(* Logix 5000 project; controller WWTP_SOLIDS_CLX vendor 1 type 14 code 54 rev 17.2; software revision 17.00; part 15 of 16 *)
(* tags used below, declared in another part *)
   Equip_Torque : ALIAS FOR I_SolidsTkDrive_Torque;
   Equip_Torque_IOFault : ALIAS FOR I_SolidsTkDrive_Torque_IOFault;
   I_P600_Fault : ALIAS FOR Local:3:I.DATA.1;
   I_P600_Fault_IOFault : ALIAS FOR Local:3:I.Fault.1;
   I_P600_InAuto : ALIAS FOR Local:3:I.Data.4;
   I_P600_InAuto_IOFault : ALIAS FOR Local:3:I.Fault.4;
   I_P600_RunFdbk : ALIAS FOR Local:3:I.Data.2;
   I_P600_RunFdbk_IOFault : ALIAS FOR Local:3:I.Fault.2;
   I_P602_Fault : ALIAS FOR Local:3:I.Data.9;
   I_P602_Fault_IOFault : ALIAS FOR Local:3:I.Fault.9;
   I_P602_InAuto : ALIAS FOR Local:3:I.Data.7;
   I_P602_InAuto_IOFault : ALIAS FOR Local:3:I.Fault.7;
   I_P602_RunFdbk : ALIAS FOR Local:3:I.Data.8;
   I_P602_RunFdbk_IOFault : ALIAS FOR Local:3:I.Fault.8;
   I_PV600_CloseLS : ALIAS FOR Local:3:I.Data.14;
   I_PV600_CloseLS_IOFault : ALIAS FOR Local:3:I.Fault.14;
   I_PV600_InAuto : ALIAS FOR Local:3:I.Data.0;
   I_PV600_InAuto_IOFault : ALIAS FOR Local:3:I.Fault.0;
   I_PV600_OpenLS : ALIAS FOR Local:3:I.Data.13;
   I_PV600_OpenLS_IOFault : ALIAS FOR Local:3:I.Fault.13;
   O_P600_Out_Run : ALIAS FOR Local:4:O.Data.1;   // P-600 Start/Stop
   O_P602_Out_Run : ALIAS FOR Local:4:O.Data.3;   // P-602 Start/Stop
   O_PV600_Close : ALIAS FOR Local:4:O.Data.5;   // P-600 Close
   O_PV600_Open : ALIAS FOR Local:4:O.Data.4;   // P-600 Open
   PLC_Device_ResetPB : BOOL;   // Site Wide Device Reset Push Button
   PLC_Simulation : BOOL;   // Application running IN SIMULATION
   SolidsTk_Lv_Ain : P_AIn;   // Solids Storage Tank Level Indication (LIT-603) 0-20 Ft
   WAS_StorageTkLv_Ain : P_AIn;   // WAS Storage Tank Level Indication (LIT-605) 0-20 Ft
(* SolidsTk01_Drive, continued *)

ROUTINE A02_Drive_FBD   (* function block diagram *)
   SHEET 1   // Motor
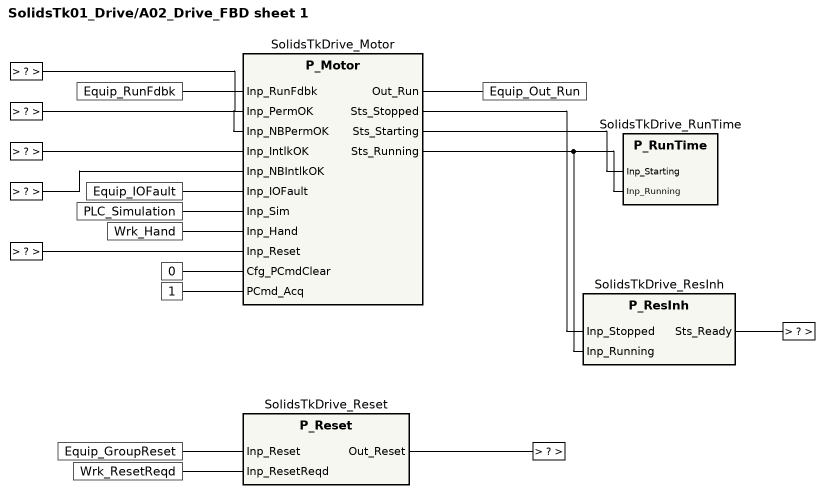
   SolidsTkDrive_Reset : P_Reset(Inp_Reset := Equip_GroupReset, Inp_ResetReqd := Wrk_ResetReqd);
   WIRE(?) := SolidsTkDrive_Reset.Out_Reset;
   SolidsTkDrive_ResInh : P_ResInh(Inp_Stopped := SolidsTkDrive_Motor.Sts_Stopped {feedback}, Inp_Running := SolidsTkDrive_Motor.Sts_Running {feedback});
   WIRE(?) := SolidsTkDrive_ResInh.Sts_Ready;
   SolidsTkDrive_Motor : P_Motor(Inp_RunFdbk := Equip_RunFdbk, Inp_PermOK := WIRE(?), Inp_NBPermOK := WIRE(?), Inp_IntlkOK := WIRE(?), Inp_NBIntlkOK := WIRE(?), Inp_IOFault := Equip_IOFault, Inp_Sim := PLC_Simulation, Inp_Hand := Wrk_Hand, Inp_Reset := WIRE(?), Cfg_PCmdClear := 0, PCmd_Acq := 1);
   Equip_Out_Run := SolidsTkDrive_Motor.Out_Run;
   SolidsTkDrive_RunTime : P_RunTime(Inp_Starting := SolidsTkDrive_Motor.Sts_Starting, Inp_Running := SolidsTkDrive_Motor.Sts_Running);
   SHEET 2   // Permissives
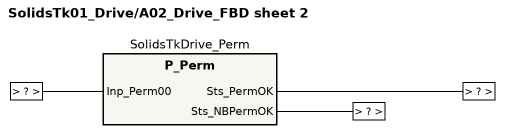
   SolidsTkDrive_Perm : P_Perm(Inp_Perm00 := WIRE(?));
   WIRE(?) := SolidsTkDrive_Perm.Sts_NBPermOK;
   WIRE(?) := SolidsTkDrive_Perm.Sts_PermOK;
   SHEET 3   // Interlocks
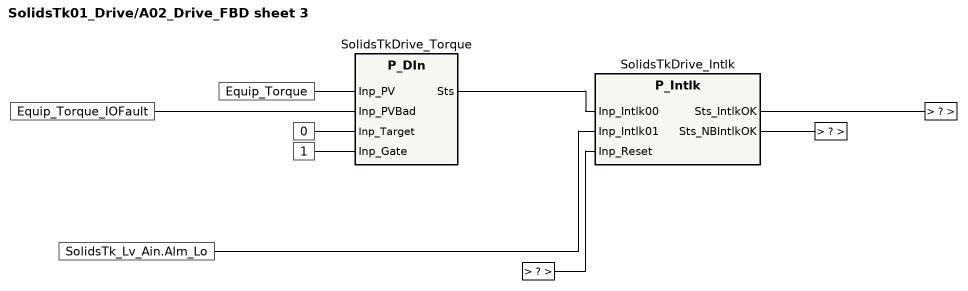
   SolidsTkDrive_Torque : P_DIn(Inp_PV := Equip_Torque, Inp_PVBad := Equip_Torque_IOFault, Inp_Target := 0, Inp_Gate := 1);
   SolidsTkDrive_Intlk : P_Intlk(Inp_Intlk00 := SolidsTkDrive_Torque.Sts, Inp_Intlk01 := SolidsTk_Lv_Ain.Alm_Lo, Inp_Reset := WIRE(?));
   WIRE(?) := SolidsTkDrive_Intlk.Sts_NBIntlkOK;
   WIRE(?) := SolidsTkDrive_Intlk.Sts_IntlkOK;
END_ROUTINE

ROUTINE Main   (* ladder *)
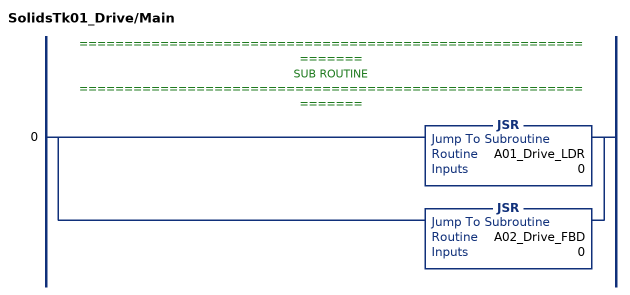
   // ===============================================================
   // SUB ROUTINE
   // ===============================================================
   0: [JSR(A01_Drive_LDR,0) ,JSR(A02_Drive_FBD,0) ];
END_ROUTINE
END_PROGRAM

PROGRAM SolidsTk01ToFilterPress_Pump602   (* main routine Main *)
VAR
   Equip_Fault : ALIAS FOR I_P602_Fault;
   Equip_Fault_IOFault : ALIAS FOR I_P602_Fault_IOFault;
   Equip_GroupReset : ALIAS FOR PLC_Device_ResetPB;
   Equip_InAuto : ALIAS FOR I_P602_InAuto;
   Equip_InAuto_IOFault : ALIAS FOR I_P602_InAuto_IOFault;
   Equip_Intlk : ALIAS FOR P602_Intlk;
   Equip_IOFault : BOOL;
   Equip_Motor : ALIAS FOR P602_Motor;
   Equip_Out_Run : ALIAS FOR O_P602_Out_Run;
   Equip_RunFdbk : ALIAS FOR I_P602_RunFdbk;
   Equip_RunFdbk_IOFault : ALIAS FOR I_P602_RunFdbk_IOFault;
   Wrk_Hand : BOOL;
   Wrk_ResetReqd : BOOL;
   Wrk_ResetRequired : BOOL;
END_VAR

ROUTINE A01_Pump_LDR   (* ladder *)
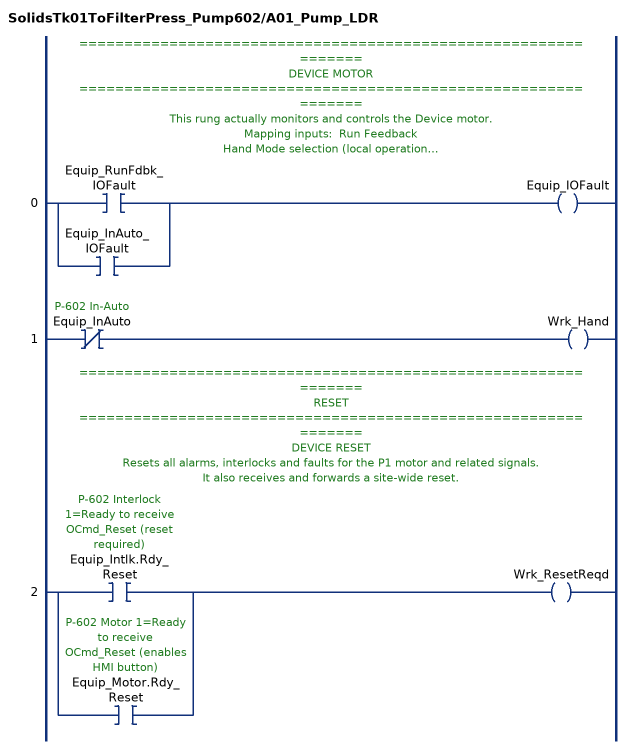
   // ===============================================================
   // DEVICE MOTOR
   // ===============================================================
   // This rung actually monitors and controls the Device motor.
   // Mapping inputs:  Run Feedback
   // Hand Mode selection (local operation)
   // Permissive OK
   // Protective’s OK,
   // I/O Fault signals
   // Pump Reset (above)
   // DEVICE
   // Output Mapping: Starter output
   0: [XIC(Equip_RunFdbk_IOFault) ,XIC(Equip_InAuto_IOFault) ]OTE(Equip_IOFault);
   1: XIO(Equip_InAuto)OTE(Wrk_Hand);
   // ===============================================================
   // RESET
   // ===============================================================
   // DEVICE RESET
   // Resets all alarms, interlocks and faults for the P1 motor and related signals.
   // It also receives and forwards a site-wide reset.
   2: [XIC(Equip_Intlk.Rdy_Reset) ,XIC(Equip_Motor.Rdy_Reset) ]OTE(Wrk_ResetReqd);
END_ROUTINE

ROUTINE A02_Pump_FBD   (* function block diagram *)
   SHEET 1   // Motor
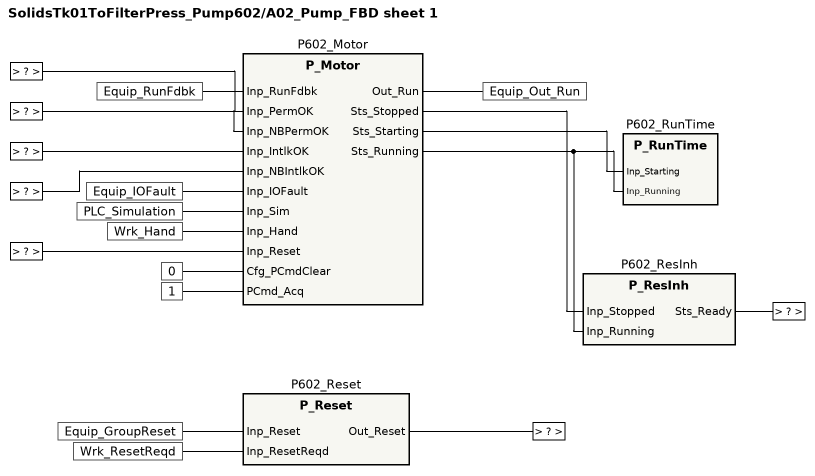
   P602_Reset : P_Reset(Inp_Reset := Equip_GroupReset, Inp_ResetReqd := Wrk_ResetReqd);
   WIRE(?) := P602_Reset.Out_Reset;
   P602_ResInh : P_ResInh(Inp_Stopped := P602_Motor.Sts_Stopped {feedback}, Inp_Running := P602_Motor.Sts_Running {feedback});
   WIRE(?) := P602_ResInh.Sts_Ready;
   P602_Motor : P_Motor(Inp_RunFdbk := Equip_RunFdbk, Inp_PermOK := WIRE(?), Inp_NBPermOK := WIRE(?), Inp_IntlkOK := WIRE(?), Inp_NBIntlkOK := WIRE(?), Inp_IOFault := Equip_IOFault, Inp_Sim := PLC_Simulation, Inp_Hand := Wrk_Hand, Inp_Reset := WIRE(?), Cfg_PCmdClear := 0, PCmd_Acq := 1);
   Equip_Out_Run := P602_Motor.Out_Run;
   P602_RunTime : P_RunTime(Inp_Starting := P602_Motor.Sts_Starting, Inp_Running := P602_Motor.Sts_Running);
   SHEET 2   // Permissives / Interlocks
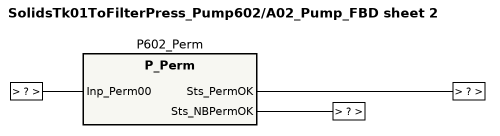
   P602_Perm : P_Perm(Inp_Perm00 := WIRE(?));
   WIRE(?) := P602_Perm.Sts_NBPermOK;
   WIRE(?) := P602_Perm.Sts_PermOK;
   SHEET 3   // Interlocks
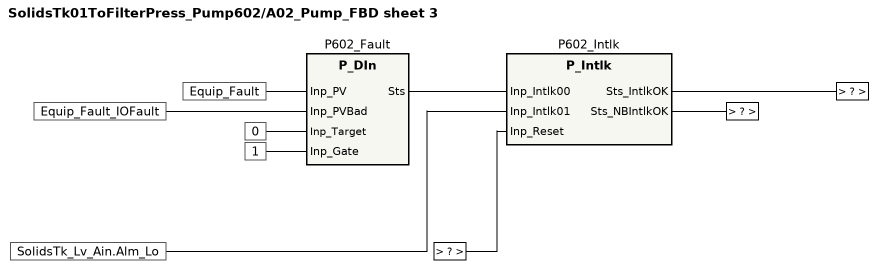
   P602_Fault : P_DIn(Inp_PV := Equip_Fault, Inp_PVBad := Equip_Fault_IOFault, Inp_Target := 0, Inp_Gate := 1);
   P602_Intlk : P_Intlk(Inp_Intlk00 := P602_Fault.Sts, Inp_Intlk01 := SolidsTk_Lv_Ain.Alm_Lo, Inp_Reset := WIRE(?));
   WIRE(?) := P602_Intlk.Sts_NBIntlkOK;
   WIRE(?) := P602_Intlk.Sts_IntlkOK;
END_ROUTINE

ROUTINE Main   (* ladder *)
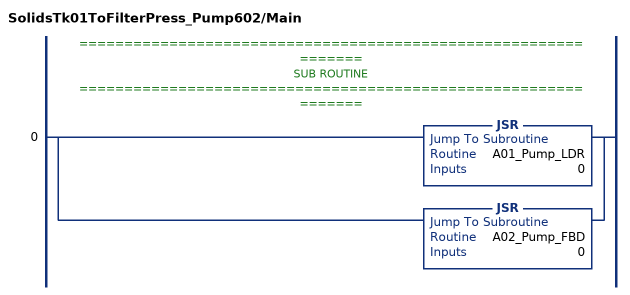
   // ===============================================================
   // SUB ROUTINE
   // ===============================================================
   0: [JSR(A01_Pump_LDR,0) ,JSR(A02_Pump_FBD,0) ];
END_ROUTINE
END_PROGRAM

PROGRAM WAS_HoldTkValve600   (* main routine Main *)
VAR
   Equip_Close : ALIAS FOR O_PV600_Close;
   Equip_CloseLS : ALIAS FOR I_PV600_CloseLS;
   Equip_CloseLS_IOFault : ALIAS FOR I_PV600_CloseLS_IOFault;
   Equip_GroupReset : ALIAS FOR PLC_Device_ResetPB;
   Equip_InAuto : ALIAS FOR I_PV600_InAuto;
   Equip_InAuto_IOFault : ALIAS FOR I_PV600_InAuto_IOFault;
   Equip_IOFault : BOOL;
   Equip_Open : ALIAS FOR O_PV600_Open;
   Equip_OpenLS : ALIAS FOR I_PV600_OpenLS;
   Equip_OpenLS_IOFault : ALIAS FOR I_PV600_OpenLS_IOFault;
   Equip_Valve : ALIAS FOR PV600;
   Wrk_Hand : BOOL;
   Wrk_ResetReqd : BOOL;
   Wrk_ResetRequired : BOOL;
END_VAR

ROUTINE A01_Valve_LDR   (* ladder *)
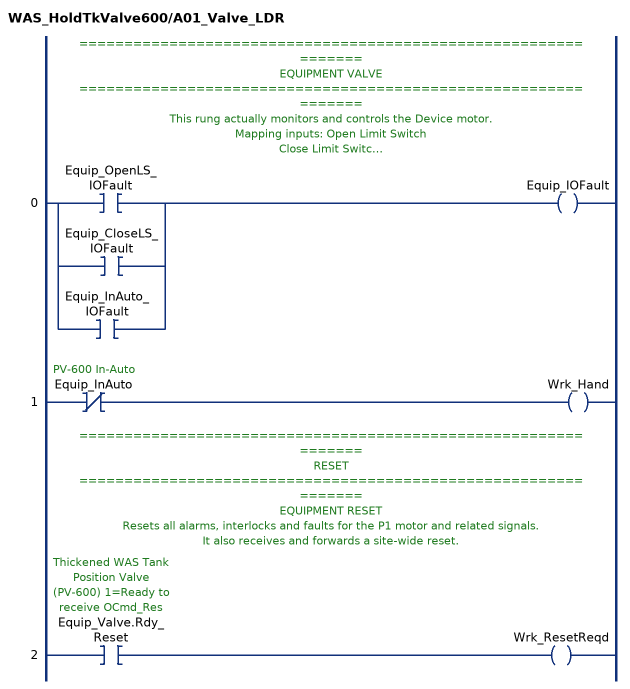
   // ===============================================================
   // EQUIPMENT VALVE
   // ===============================================================
   // This rung actually monitors and controls the Device motor.
   // Mapping inputs: Open Limit Switch
   // Close Limit Switch
   // Hand Mode selection (local operation)
   // Open Permissive OK
   // Close Permissive OK
   // I/O Fault signals
   // Pump Reset (above)
   // EQUIPMENT
   // Output Mapping: Open output
   // Close output
   0: [XIC(Equip_OpenLS_IOFault) ,XIC(Equip_CloseLS_IOFault) ,XIC(Equip_InAuto_IOFault) ]OTE(Equip_IOFault);
   1: XIO(Equip_InAuto)OTE(Wrk_Hand);
   // ===============================================================
   // RESET
   // ===============================================================
   // EQUIPMENT RESET
   // Resets all alarms, interlocks and faults for the P1 motor and related signals.
   // It also receives and forwards a site-wide reset.
   2: XIC(Equip_Valve.Rdy_Reset)OTE(Wrk_ResetReqd);
END_ROUTINE

ROUTINE A02_Valve_FBD   (* function block diagram *)
   SHEET 1   // Valve
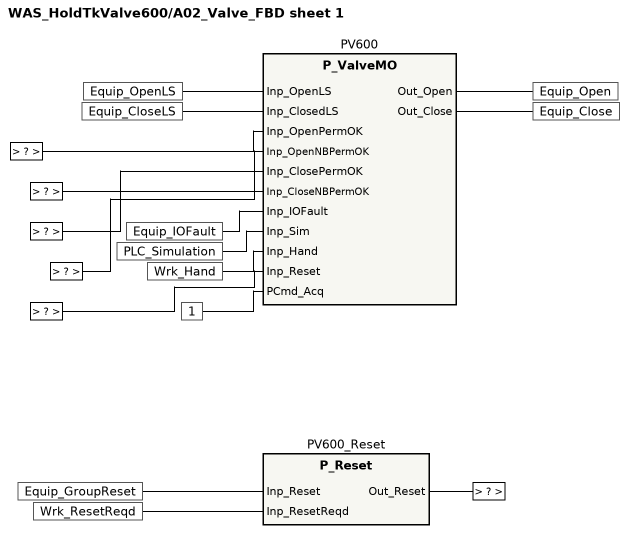
   PV600_Reset : P_Reset(Inp_Reset := Equip_GroupReset, Inp_ResetReqd := Wrk_ResetReqd);
   WIRE(?) := PV600_Reset.Out_Reset;
   PV600 : P_ValveMO(Inp_OpenLS := Equip_OpenLS, Inp_ClosedLS := Equip_CloseLS, Inp_OpenPermOK := WIRE(?), Inp_OpenNBPermOK := WIRE(?), Inp_ClosePermOK := WIRE(?), Inp_CloseNBPermOK := WIRE(?), Inp_IOFault := Equip_IOFault, Inp_Sim := PLC_Simulation, Inp_Hand := Wrk_Hand, Inp_Reset := WIRE(?), PCmd_Acq := 1);
   Equip_Open := PV600.Out_Open;
   Equip_Close := PV600.Out_Close;
   SHEET 2   // Open Permissives
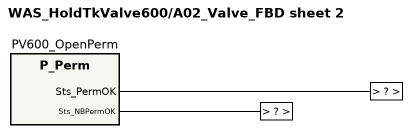
   PV600_OpenPerm : P_Perm();
   WIRE(?) := PV600_OpenPerm.Sts_NBPermOK;
   WIRE(?) := PV600_OpenPerm.Sts_PermOK;
   SHEET 3   // Close Permissives
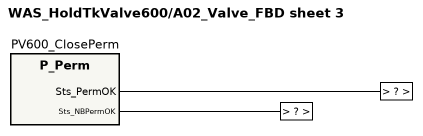
   PV600_ClosePerm : P_Perm();
   WIRE(?) := PV600_ClosePerm.Sts_NBPermOK;
   WIRE(?) := PV600_ClosePerm.Sts_PermOK;
END_ROUTINE

ROUTINE Main   (* ladder *)
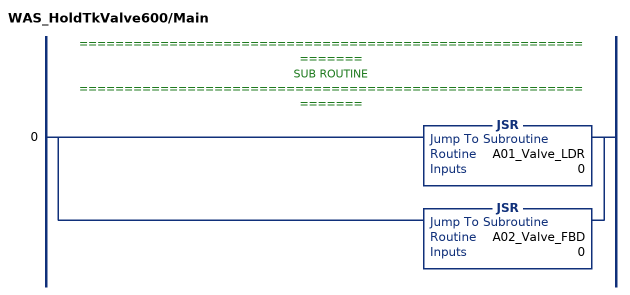
   // ===============================================================
   // SUB ROUTINE
   // ===============================================================
   0: [JSR(A01_Valve_LDR,0) ,JSR(A02_Valve_FBD,0) ];
END_ROUTINE
END_PROGRAM

PROGRAM WAS_StorageTk_ToSolidsTk01_Pump600   (* main routine Main *)
VAR
   Equip_Fault : ALIAS FOR I_P600_Fault;
   Equip_Fault_IOFault : ALIAS FOR I_P600_Fault_IOFault;
   Equip_GroupReset : ALIAS FOR PLC_Device_ResetPB;
   Equip_InAuto : ALIAS FOR I_P600_InAuto;
   Equip_InAuto_IOFault : ALIAS FOR I_P600_InAuto_IOFault;
   Equip_Intlk : ALIAS FOR P600_Intlk;
   Equip_IOFault : BOOL;
   Equip_Motor : ALIAS FOR P600_Motor;
   Equip_Out_Run : ALIAS FOR O_P600_Out_Run;
   Equip_RunFdbk : ALIAS FOR I_P600_RunFdbk;
   Equip_RunFdbk_IOFault : ALIAS FOR I_P600_RunFdbk_IOFault;
   Wrk_Hand : BOOL := 1;
   Wrk_ResetReqd : BOOL;
   Wrk_ResetRequired : BOOL;
END_VAR

ROUTINE A01_Pump_LDR   (* ladder *)
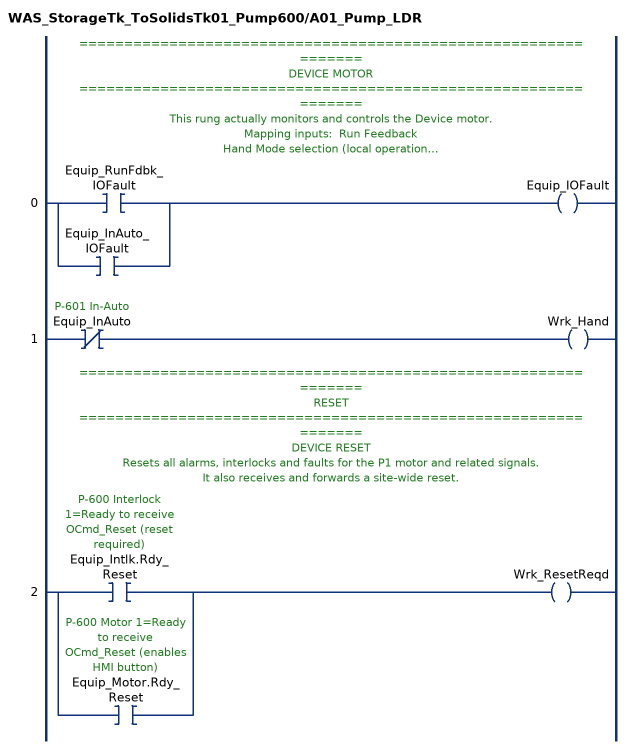
   // ===============================================================
   // DEVICE MOTOR
   // ===============================================================
   // This rung actually monitors and controls the Device motor.
   // Mapping inputs:  Run Feedback
   // Hand Mode selection (local operation)
   // Permissive OK
   // Protective’s OK,
   // I/O Fault signals
   // Pump Reset (above)
   // DEVICE
   // Output Mapping: Starter output
   0: [XIC(Equip_RunFdbk_IOFault) ,XIC(Equip_InAuto_IOFault) ]OTE(Equip_IOFault);
   1: XIO(Equip_InAuto)OTE(Wrk_Hand);
   // ===============================================================
   // RESET
   // ===============================================================
   // DEVICE RESET
   // Resets all alarms, interlocks and faults for the P1 motor and related signals.
   // It also receives and forwards a site-wide reset.
   2: [XIC(Equip_Intlk.Rdy_Reset) ,XIC(Equip_Motor.Rdy_Reset) ]OTE(Wrk_ResetReqd);
END_ROUTINE

ROUTINE A02_Pump_FBD   (* function block diagram *)
   SHEET 1   // Motor
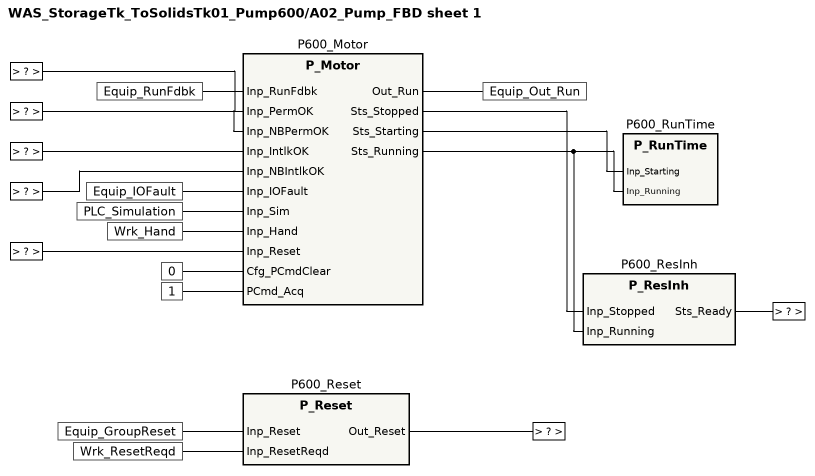
   P600_Reset : P_Reset(Inp_Reset := Equip_GroupReset, Inp_ResetReqd := Wrk_ResetReqd);
   WIRE(?) := P600_Reset.Out_Reset;
   P600_ResInh : P_ResInh(Inp_Stopped := P600_Motor.Sts_Stopped {feedback}, Inp_Running := P600_Motor.Sts_Running {feedback});
   WIRE(?) := P600_ResInh.Sts_Ready;
   P600_Motor : P_Motor(Inp_RunFdbk := Equip_RunFdbk, Inp_PermOK := WIRE(?), Inp_NBPermOK := WIRE(?), Inp_IntlkOK := WIRE(?), Inp_NBIntlkOK := WIRE(?), Inp_IOFault := Equip_IOFault, Inp_Sim := PLC_Simulation, Inp_Hand := Wrk_Hand, Inp_Reset := WIRE(?), Cfg_PCmdClear := 0, PCmd_Acq := 1);
   Equip_Out_Run := P600_Motor.Out_Run;
   P600_RunTime : P_RunTime(Inp_Starting := P600_Motor.Sts_Starting, Inp_Running := P600_Motor.Sts_Running);
   SHEET 2   // Permissives / Interlocks
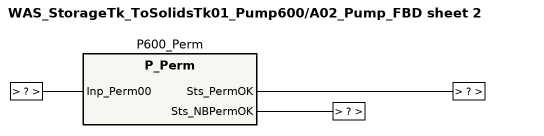
   P600_Perm : P_Perm(Inp_Perm00 := WIRE(?));
   WIRE(?) := P600_Perm.Sts_NBPermOK;
   WIRE(?) := P600_Perm.Sts_PermOK;
   SHEET 3   // Interlocks
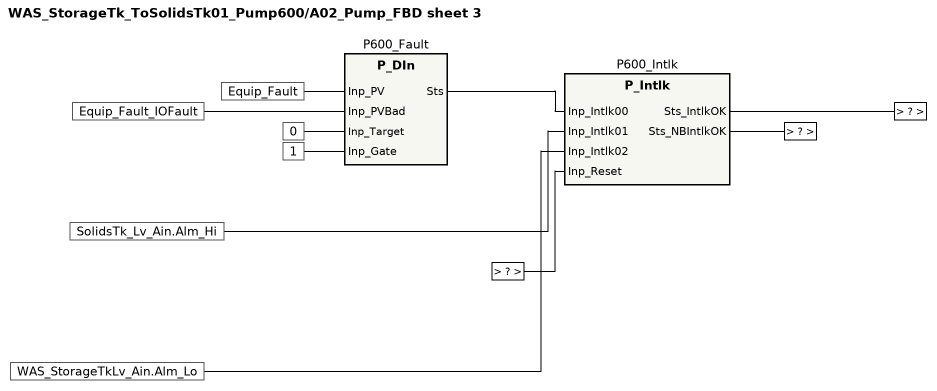
   P600_Fault : P_DIn(Inp_PV := Equip_Fault, Inp_PVBad := Equip_Fault_IOFault, Inp_Target := 0, Inp_Gate := 1);
   P600_Intlk : P_Intlk(Inp_Intlk00 := P600_Fault.Sts, Inp_Intlk01 := SolidsTk_Lv_Ain.Alm_Hi, Inp_Intlk02 := WAS_StorageTkLv_Ain.Alm_Lo, Inp_Reset := WIRE(?));
   WIRE(?) := P600_Intlk.Sts_NBIntlkOK;
   WIRE(?) := P600_Intlk.Sts_IntlkOK;
END_ROUTINE
